{attribute addProperty BoxType "EP5101-0002-0016"}
{attribute addProperty Id "ENC_Status_compactAT %I*ENC_Status_compact_18E0726F4860ENC_Control_compactAT %Q*ENC_Control_compact_3146A3B23240WcStateAT %I*WcState_F855686C1620InfoDataAT %I*InfoData_BC63D37F80100"}
{attribute addProperty CRC "3493233234"}
{attribute addProperty SizeInBites "176"}
{attribute addProperty SizeInBytes "22"}
TYPE EP5101_F338D8E4 :
STRUCT
	{attribute addProperty Name "ENC_Status_compact"}
	ENC_Status_compact : ENC_Status_compact_18E0726F;
	{attribute addProperty Name "ENC_Control_compact"}
	ENC_Control_compact : ENC_Control_compact_3146A3B2;
	{attribute addProperty Name "WcState"}
	WcState : WcState_F855686C;
	{attribute addProperty Name "InfoData"}
	InfoData : InfoData_BC63D37F;
END_STRUCT
END_TYPE

(* stored: Version 1.2.0.0, ProductVersion 3.1.4024.9
   DUT EP5101_F338D8E4: Id {96994c1c-37d3-4235-aea2-38a1d4007b4a} *)
